TYPE udt_SRxx_ToUI_20260122 :
STRUCT
	DiscreteImage : udt_SRxx_DiscreteImage;
END_STRUCT
END_TYPE

(* stored: Version 1.1.0.1, ProductVersion 3.1.4024.12
   DUT udt_SRxx_ToUI_20260122: Id {83a14239-9182-4d26-bf71-b27e868b0f2d} *)
